FUNCTION fun_Modulo : LREAL
VAR_INPUT
	fVar: LREAL;
	fModulo: LREAL:=360.0;

END_VAR
VAR
END_VAR

fun_Modulo:=fVar;
IF fun_Modulo>0 THEN;
	WHILE fun_Modulo>=fModulo DO
		fun_Modulo:=fun_Modulo-fModulo;
	END_WHILE
ELSE;
	WHILE fun_Modulo<0 DO
		fun_Modulo:=fun_Modulo+fModulo;
	END_WHILE	
END_IF

END_FUNCTION

(* stored: Version 1.1.0.1, ProductVersion 3.1.4024.12
   POU fun_Modulo: Id {b7613cba-50f9-4fff-b7c4-a1abfca5fd37}, SpecialFunc None *)
